(* Schneider Machine Expert - Basic project tank_level_v6_TM221CE16T, file version 3.0.0.0 *)
(* ProjectInformations: Name=Tank Level Control v6 *)

HARDWARE
  Cpu 0: TM221CE16T
  ModuleExtensionObject 0: TM3AI4/G
  EthernetConfiguration: NetworkName=M221, IpAllocationMode=FixedAddress, IpAddress=0.0.0.0, SubnetMask=0.0.0.0
  SerialLineConfiguration: Baud=Baud19200, Parity=ParityEven, DataBits=DataBits8, StopBits=StopBits1, PhysicalMedium=PhysicalMediumRs485, TransmissionMode=TransmissionModeModbusRtu, SlaveId=1, Addressing=SlaveAddressing
  MastTask: UsePeriodScanMode=false, PeriodScan=100
  FastTask: Period=255
  CpuBehavior: StartingMode=StartAsPreviousState, AutoSaveRamOnEeprom=true, WatchdogPeriod=250

SYMBOLS  (address, symbol, comment, settings)
  %IW1.0    TANK_LEVEL  [Type=Type_4_20mA, Scope=Scope_Customized, Minimum=300, Maximum=3000]

POU Tank Level Control
  (* SectionNumber=0 *)

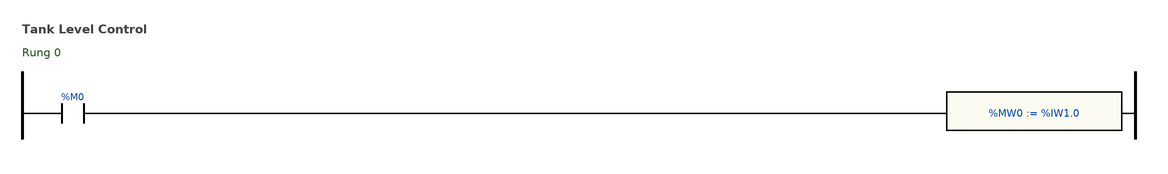

// Rung 0
  LD %M0
  [ %MW0 := %IW1.0 ]      (* TANK_LEVEL *)
  // as ST:
  //   IF %M0 THEN %MW0 := TANK_LEVEL; END_IF;
